FUNCTION_BLOCK RampCtrl
VAR_INPUT
	Target: REAL := 0;
END_VAR
VAR_OUTPUT
	MomentarySetpoint: REAL := 0;
END_VAR
VAR
	Initialized: BOOL := FALSE;
	Velocity: REAL := 1;
	CycleTimeSeconds: REAL := 0;
	Direction: REAL;
	SetpointReached: BOOL := FALSE;
END_VAR

IF NOT Initialized THEN  // initialization
	CycleTimeSeconds := UDINT_TO_REAL(_TaskInfo[GETCURTASKINDEXEX()].CycleTime) / 10_000_000;
	Initialized := TRUE;
END_IF

SetpointReached := (Target = MomentarySetpoint);

IF NOT SetpointReached THEN
	Direction := (Target - MomentarySetpoint) / ABS(Target - MomentarySetpoint);
	MomentarySetpoint := MomentarySetpoint + Direction * Velocity * CycleTimeSeconds;
	IF Direction < 0 THEN
		MomentarySetpoint := MAX(Target, MomentarySetpoint);
	ELSE
		MomentarySetpoint := MIN(Target, MomentarySetpoint);
	END_IF
END_IF

END_FUNCTION_BLOCK

(* stored: Version 1.1.0.1, ProductVersion 3.1.4024.15
   POU RampCtrl: Id {81290241-ad53-4ddf-bdcb-a240bb10f9af}, SpecialFunc None *)
